// TIA Portal V20 export
FUNCTION_BLOCK "FB_Pressures"   // FB440, SCL
{ S7_Optimized_Access := 'TRUE' }
// stored: AutoNumber false, IsIECCheckEnabled true, MemoryReserve 100, SetENOAutomatically false
   VAR
      sTimeOutAirDryer : TON_TIME;
      sTimerMachineInDelay : TON_TIME;
      sTimeMachineReadyDelay { S7_SetPoint := 'True'} : TON_TIME;
      sAirInletPressureCtrl { S7_SetPoint := 'True'} : "FB_AnalogInputThreshold";
      sOverpressureScaleZ_Ctrl { S7_SetPoint := 'True'} : "FB_AnalogInputThreshold";
      sOverpressureOpticalPathCtrl { S7_SetPoint := 'True'} : "FB_AnalogInputThreshold";
      sOverpressureLaserHeadCtrl { S7_SetPoint := 'True'} : "FB_AnalogInputThreshold";
      sOverpressureAxisX_Y_Ctrl { S7_SetPoint := 'True'} : "FB_AnalogInputThreshold";
   END_VAR
   VAR CONSTANT
      TIME_OUT_DRYER : Time := T#15S;   // Output short pulse blinking
      TIME_MACHINE_IN_DELAY : Time := T#2S;   // Output short pulse blinking
      OVER_PRESSURE_VALVE_DELAY : Time := T#1S;
      TIME_WAIT_PRESSURE : Time := T#5s;
   END_VAR
BEGIN
   REGION Description header 
       //==================================================================================
       // POSALUX Swiss SA / (C) Copyright 2024
       //----------------------------------------------------------------------------------
       // Title: Management of the pressures of the machine
       // Comment/Function: 
       //
       // Author: Gowsigan SRITHARAN
       // Engineering: TIA Portal v19
       // 
       //----------------------------------------------------------------------------------
       // Change log table:
       // Version  | Date     | Expert in charge | Changes applied
       // ---------|----------|------------------|------------------------------------
       // 00.00.01 | 20250516 | GSR              | First released version
       // ==================================================================================
   END_REGION

   //==================================================================================
   ///////////////////////////////// TECHNICAL TOWER //////////////////////////////////
   // =================================================================================
   REGION Dryer 
       #sTimeOutAirDryer(IN := "DB_PowerOn".sMachineReadySoft AND NOT "DB_DigitalInputs".sAirDryerOK.sSWStatus,
                         PT := #TIME_OUT_DRYER,
                         Q => "LBP_AlarmMsgs".UserA[4].A70UUxx[9]);
   END_REGION

   REGION Air Inlet Pressure
       #sAirInletPressureCtrl(iActualValue:= "DB_AnalogInputs".sInletAirPressure.sSWRealValue,
                              iStartDelay:= "DB_PowerOn".sTimeMachineReadyDelay.Q,
                              ioAlarmMin:= "LBP_AlarmMsgs".UserA[06].A70UUxx[40],
                              ioWarningMin:= "LBP_AlarmMsgs".UserA[07].A70UUxx[40],
                              ioWarningMax:= "LBP_AlarmMsgs".UserA[07].A70UUxx[41],
                              ioAlarmMax:= "LBP_AlarmMsgs".UserA[06].A70UUxx[41],
                              oDataAction=> "DB_AnalogInputAction".Inlet_Air_Pressure,
                              iDataPLC := "DB_AnalogInputDataPLC".Inlet_Air_Pressure,
                              iDataHMI:= "DB_AnalogInputDataHMI".Inlet_Air_Pressure);
   END_REGION

   REGION Output pressure general air
       "DB_DigitalOutputs".sGeneralAirValve.sSWStatus := "DB_PowerOn".sMachineReadySoft;

   END_REGION

   REGION Alarm air pressure
      // pneumatic branching module
       IF "DB_PowerOn".sTimeMachineReadyDelay.Q AND NOT "DB_DigitalInputs".sAirPressureCtrl.sSWStatus THEN
          "LBP_AlarmMsgs".UserA[00].A70UUxx[05] := TRUE;
      END_IF;
   END_REGION

   //==================================================================================
   ///////////////////////////////////// MACHINE //////////////////////////////////////
   //==================================================================================
   REGION Overpressure Scale Z
       #sOverpressureScaleZ_Ctrl(iActualValue:= "DB_AnalogInputs".sZLAxisOverpressure.sSWRealValue,
                                 iStartDelay:= "DB_PowerOn".sTimeMachineReadyDelay.Q,
                                 ioAlarmMin:= "LBP_AlarmMsgs".UserA[06].A70UUxx[42],
                                 ioWarningMin:= "LBP_AlarmMsgs".UserA[07].A70UUxx[42],
                                 ioWarningMax:= "LBP_AlarmMsgs".UserA[07].A70UUxx[43],
                                 ioAlarmMax:= "LBP_AlarmMsgs".UserA[06].A70UUxx[43],
                                 oDataAction=> "DB_AnalogInputAction".ZL_Axis_Overpressure,
                                 iDataPLC := "DB_AnalogInputDataPLC".ZL_Axis_Overpressure,
                                 iDataHMI:= "DB_AnalogInputDataHMI".ZL_Axis_Overpressure);
   END_REGION

   REGION Overpressure Optical path
       #sOverpressureOpticalPathCtrl(iActualValue := "DB_AnalogInputs".sOpticalPathOverpressure.sSWRealValue,
                                     iStartDelay := "DB_PowerOn".sTimeMachineReadyDelay.Q,
                                     ioAlarmMin := "LBP_AlarmMsgs".UserA[06].A70UUxx[44],
                                     ioWarningMin := "LBP_AlarmMsgs".UserA[07].A70UUxx[44],
                                     ioWarningMax := "LBP_AlarmMsgs".UserA[07].A70UUxx[45],
                                     ioAlarmMax := "LBP_AlarmMsgs".UserA[06].A70UUxx[45],
                                     oDataAction=> "DB_AnalogInputAction".Optical_Path_Overpressure,
                                     iDataPLC := "DB_AnalogInputDataPLC".Optical_Path_Overpressure,
                                     iDataHMI := "DB_AnalogInputDataHMI".Optical_Path_Overpressure);
   END_REGION

   REGION Overpressure Laser Head
       #sOverpressureLaserHeadCtrl(iActualValue := "DB_AnalogInputs".sLaserHeadOverpressure.sSWRealValue,
                                   iStartDelay := "DB_PowerOn".sTimeMachineReadyDelay.Q,
                                   ioAlarmMin := "LBP_AlarmMsgs".UserA[06].A70UUxx[46],
                                   ioWarningMin := "LBP_AlarmMsgs".UserA[07].A70UUxx[46],
                                   ioWarningMax := "LBP_AlarmMsgs".UserA[07].A70UUxx[47],
                                   ioAlarmMax := "LBP_AlarmMsgs".UserA[06].A70UUxx[47],
                                   oDataAction=> "DB_AnalogInputAction".Laser_Head_Overpressure,
                                   iDataPLC := "DB_AnalogInputDataPLC".Laser_Head_Overpressure,
                                   iDataHMI := "DB_AnalogInputDataHMI".Laser_Head_Overpressure);
   END_REGION

   REGION Overpressure Axis X and Y
       #sOverpressureAxisX_Y_Ctrl(iActualValue := "DB_AnalogInputs".sXYAxisOverpressure.sSWRealValue,
                                  iStartDelay := "DB_PowerOn".sTimeMachineReadyDelay.Q,
                                  ioAlarmMin := "LBP_AlarmMsgs".UserA[06].A70UUxx[48],
                                  ioWarningMin := "LBP_AlarmMsgs".UserA[07].A70UUxx[48],
                                  ioWarningMax := "LBP_AlarmMsgs".UserA[07].A70UUxx[49],
                                  ioAlarmMax := "LBP_AlarmMsgs".UserA[06].A70UUxx[49],
                                  oDataAction=> "DB_AnalogInputAction".XY_Axis_Overpressure,
                                  iDataPLC := "DB_AnalogInputDataPLC".XY_Axis_Overpressure,
                                  iDataHMI := "DB_AnalogInputDataHMI".XY_Axis_Overpressure);
   END_REGION

   REGION Brake Pressure Ctrl 
       // Reset Channel Feed Disable
       IF "DB_McpKeyboardSignals".sAlarmReset.sKeySWStatus THEN
           "LBP_AlarmMsgs".Chan[1].FDD[9] := FALSE;
       END_IF;

       // X Axis
       IF "DB_PowerOn".sMachinePower
           AND ("LBP_Axis01_X".E_TReqMinus OR "LBP_Axis01_X".E_TReqPlus)
           AND NOT "DB_DigitalInputs".sX_AxisBrakePressCtrl.sSWStatus THEN
           "LBP_AlarmMsgs".UserA[00].A70UUxx[06] := TRUE;
           "LBP_AlarmMsgs".Chan[1].FDD[9] := TRUE;
       END_IF;

       // Y Axis
       IF "DB_PowerOn".sMachinePower
           AND ("LBP_Axis02_Y".E_TReqMinus OR "LBP_Axis02_Y".E_TReqPlus)
           AND NOT "DB_DigitalInputs".sY_AxisBrakePressCtrl.sSWStatus THEN
           "LBP_AlarmMsgs".UserA[00].A70UUxx[07] := TRUE;
           "LBP_AlarmMsgs".Chan[1].FDD[9] := TRUE;
       END_IF;

       // B Axis
       IF "DB_PowerOn".sMachinePower
           AND ("LBP_Axis04_B".E_TReqMinus OR "LBP_Axis04_B".E_TReqPlus)
           AND NOT "DB_DigitalInputs".sB_Axis_BrakeReleasedCtrl.sSWStatus THEN
           "LBP_AlarmMsgs".UserA[00].A70UUxx[08] := TRUE;
           "LBP_AlarmMsgs".Chan[1].FDD[9] := TRUE;
       END_IF;
   END_REGION
END_FUNCTION_BLOCK
